GLOBALCONSTANTS DataPanel_MI_DI (* DataPanel Modules with medium IO density DI constants *)
  (* Standard: 61499-1; Description: Copyright (c) 2024 HR Agrartechnik GmbH This program and the accompanying materials are made available under the terms of the Eclipse Public License 2.0 which is available at https://www.eclipse.org/legal/epl-2.0/ SPDX-License-Identifier: EPL-2.0 *)
  (* Version 1.0, 2024-01-25, Franz Höpfinger, HR Agrartechnik GmbH *)
  PACKAGE DataPanel::io::MI::DI;
  VAR_GLOBAL CONSTANT
    DigitalInput_5A : DataPanel::io::MI::DI::DataPanel_MI_DI_S := (Pin := 9);
    DigitalInput_5B : DataPanel::io::MI::DI::DataPanel_MI_DI_S := (Pin := 10);
    DigitalInput_6A : DataPanel::io::MI::DI::DataPanel_MI_DI_S := (Pin := 11);
    DigitalInput_6B : DataPanel::io::MI::DI::DataPanel_MI_DI_S := (Pin := 12);
    DigitalInput_7A : DataPanel::io::MI::DI::DataPanel_MI_DI_S := (Pin := 13);
    DigitalInput_7B : DataPanel::io::MI::DI::DataPanel_MI_DI_S := (Pin := 14);
    DigitalInput_8A : DataPanel::io::MI::DI::DataPanel_MI_DI_S := (Pin := 15);
    DigitalInput_8B : DataPanel::io::MI::DI::DataPanel_MI_DI_S := (Pin := 16);
    Invalid : DataPanel::io::MI::DI::DataPanel_MI_DI_S := (Pin := 255);
  END_VAR
END_GLOBALCONSTANTS
